SUBAPPLICATION Heben_Senken_TO_QDA_PWM_OPC (* 2 Remote-Kommandos (Heben/Senken, je Subscribe+State-Publish, ODER-verknuepft mit IO-Test wie bei ILOCK_SWITCH_2_QXA_OPC) auf 1 ratiometrisches PWM-Signal (Danfoss PVEA: 25%=Senken, 50%=Neutral, 75%=Heben, Lastteiler-korrigiert) + 1 Freigabe-DO als Klick-Toggle (AX_T_FF_INIT, Default AN, per RPC-Methode aus VT und Dashboard aus-/einschaltbar - Not-Bedienung, z.B. Strassenmodus). Generisch fuer jeden PVEA-Aktor mit 2 physischen Kanaelen (links=PWM, rechts=Freigabe), Bedienung von einem Modul ohne eigenes VT. *)
  (* Standard: 61499-2 *)
  (* Version 1.4, 2026-09-20, Franz Höpfinger, Meisterschulen am Ostbahnhof, PWM_POW-Socket ergaenzt (reiner Passthrough an PWM_Mux.PWM_POW), da HebenSenken_ILOCK_QDA_PWM_OPC v1.1 PWM_POW jetzt als eigenen Socket statt intern fest 1.0 hat - jeder Aufrufer muss ihn jetzt verbinden. *)
  (* Version 1.3, 2026-09-08, Franz Höpfinger, Meisterschulen am Ostbahnhof, V1.1: IO-Test fuer Heben/Senken ergaenzt (SUBSCRIBE_TEST_HEBEN/SENKEN, ODER vor dem ILOCK), Publish-Punkte (State+Test) hinter den ILOCK verlegt (wie ILOCK_SWITCH_2_QXA_OPC), Freigabe-DO von starrem initval_AX auf AX_T_FF_INIT-Klick-Toggle per RPC-Methode umgestellt - KEIN OR nach dem Flipflop, AX_T_FF_INIT.Q ist alleinige Source of Truth fuer den Ausgang. V1.2: Freigabe-DO-Teilnetz nach MyLib::sys::DO_TOGGLE_RPC_QXA_OPC ausgelagert. V1.3: PWM/ILOCK/Mux-Teilnetz nach MyLib::sys::HebenSenken_ILOCK_QDA_PWM_OPC ausgelagert - diese SubApp ist jetzt nur noch die Zusammensetzung beider Bausteine, Schnittstelle unveraendert. *)
  PACKAGE MyLib::sys;
  IMPORT logiBUS::io::DQ::logiBUS_DO;
  IMPORT logiBUS::io::DQ::logiBUS_DO_S;
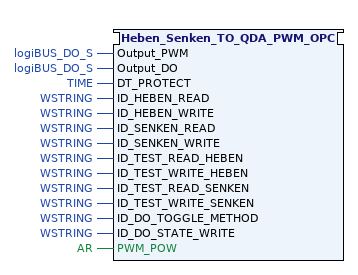
  VAR_INPUT
    Output_PWM : logiBUS::io::DQ::logiBUS_DO_S := logiBUS_DO::Invalid; (* Physischer PWM-Ausgang (linker Kanal): 25/50/75% Tastgrad, ratiometrisch *)
    Output_DO : logiBUS::io::DQ::logiBUS_DO_S := logiBUS_DO::Invalid; (* Physischer Freigabe-Ausgang (rechter Kanal): Klick-Toggle, Default AN *)
    DT_PROTECT : TIME := T#300ms; (* Schutz-Totzeit vor Richtungswechsel *)
    ID_HEBEN_READ : WSTRING; (* Echtes Funktions-Kommando Heben (Subscribe) *)
    ID_HEBEN_WRITE : WSTRING; (* Echte Funktions-Rueckmeldung Heben, HINTER dem ILOCK (Publish) *)
    ID_SENKEN_READ : WSTRING; (* Echtes Funktions-Kommando Senken (Subscribe) *)
    ID_SENKEN_WRITE : WSTRING; (* Echte Funktions-Rueckmeldung Senken, HINTER dem ILOCK (Publish) *)
    ID_TEST_READ_HEBEN : WSTRING; (* Bestehende IO-Test-Subscribe-Adresse Heben (z.B. STG2_Q0x_READ), ODER-verknuepft mit ID_HEBEN_READ vor dem ILOCK *)
    ID_TEST_WRITE_HEBEN : WSTRING; (* Bestehende IO-Test-Publish-Adresse Heben, HINTER dem ILOCK (z.B. STG2_Q0x_WRITE) *)
    ID_TEST_READ_SENKEN : WSTRING; (* Bestehende IO-Test-Subscribe-Adresse Senken, ODER-verknuepft mit ID_SENKEN_READ vor dem ILOCK *)
    ID_TEST_WRITE_SENKEN : WSTRING; (* Bestehende IO-Test-Publish-Adresse Senken, HINTER dem ILOCK *)
    ID_DO_TOGGLE_METHOD : WSTRING; (* Lokale Methodenadresse (ACTION=CREATE_METHOD) fuer den argumentlosen Freigabe-Toggle-Trigger - wird von STG1 (SoftKey-Relay) UND direkt vom OPC-Dashboard (CALL_METHOD) aufgerufen, beide Aufrufer teilen sich denselben Flipflop-Takt *)
    ID_DO_STATE_WRITE : WSTRING; (* Lokale Publish-Adresse (ACTION=WRITE) fuer den tatsaechlichen Freigabe-Zustand (AX_T_FF_INIT.Q) - wird von VT und Dashboard remote abonniert *)
  END_VAR
  SOCKETS
    PWM_POW : adapter::types::unidirectional::AR; (* PWM Power 1.0 = Maximale Power, 0.0 = Aus, 0.5 = Halb - durchgereicht an PWM_Mux.PWM_POW *)
  END_SOCKETS
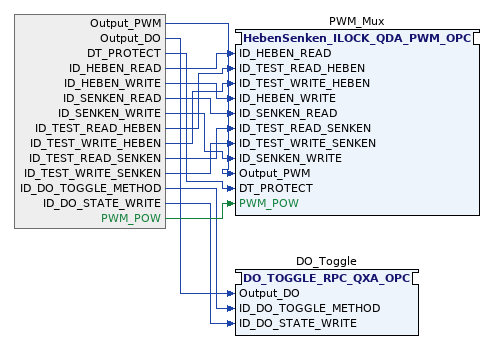
  SUBAPPS
    PWM_Mux : MyLib::sys::HebenSenken_ILOCK_QDA_PWM_OPC;
    DO_Toggle : MyLib::sys::DO_TOGGLE_RPC_QXA_OPC;
  END_SUBAPPS
  DATA_CONNECTIONS
    ID_HEBEN_READ TO PWM_Mux.ID_HEBEN_READ;
    ID_TEST_READ_HEBEN TO PWM_Mux.ID_TEST_READ_HEBEN;
    ID_TEST_WRITE_HEBEN TO PWM_Mux.ID_TEST_WRITE_HEBEN;
    ID_HEBEN_WRITE TO PWM_Mux.ID_HEBEN_WRITE;
    ID_SENKEN_READ TO PWM_Mux.ID_SENKEN_READ;
    ID_TEST_READ_SENKEN TO PWM_Mux.ID_TEST_READ_SENKEN;
    ID_TEST_WRITE_SENKEN TO PWM_Mux.ID_TEST_WRITE_SENKEN;
    ID_SENKEN_WRITE TO PWM_Mux.ID_SENKEN_WRITE;
    Output_PWM TO PWM_Mux.Output_PWM;
    DT_PROTECT TO PWM_Mux.DT_PROTECT;
    Output_DO TO DO_Toggle.Output_DO;
    ID_DO_TOGGLE_METHOD TO DO_Toggle.ID_DO_TOGGLE_METHOD;
    ID_DO_STATE_WRITE TO DO_Toggle.ID_DO_STATE_WRITE;
  END_CONNECTIONS
  ADAPTER_CONNECTIONS
    PWM_POW TO PWM_Mux.PWM_POW;
  END_CONNECTIONS
END_SUBAPPLICATION
